FUNCTION_BLOCK Disposable
VAR
END_VAR

METHOD PUBLIC Dispose
VAR_INPUT
END_VAR
__DELETE(THIS);
END_METHOD

END_FUNCTION_BLOCK

(* stored: Version 1.1.0.1, ProductVersion 3.1.4024.12
   POU Disposable: Id {f04eeb6d-b72f-43c2-a91c-3e3fca534c46}, SpecialFunc None
   Method Dispose: Id {afa659c0-7d26-4e8d-bb18-d763945e6dba} *)
